{attribute 'qualified_only'}
TYPE E_Mode :
(
    MASTER_Override :=1,
    Protection := 2,
    Maintenance := 3
);
END_TYPE

(* stored: Version 1.1.0.1, ProductVersion 3.1.4024.12
   DUT E_Mode: Id {b192f05f-9cc3-4a3c-a548-a2ff9597acb8} *)
